// TIA Portal V20 export
// export: Created 2026-07-22T09:37:46.3128458Z, ExportSetting WithDefaults, DisplayName Totally Integrated Automation Portal, DisplayVersion V20, DisplayName TIA Portal Openness, DisplayVersion V20, DisplayName TIA Portal Version Control Interface, DisplayVersion V20, DisplayName STEP 7 Professional, DisplayVersion V20, DisplayName STEP 7 Safety, DisplayVersion V20, DisplayName WinCC Basic/Comfort/Advanced, DisplayVersion V20, DisplayName WinCC Professional, DisplayVersion V20, DisplayName WinCC Unified, DisplayVersion V20
TYPE "Valve_IO"
// stored: IsFailsafeCompliant false
   STRUCT
      Configured : Bool;
      OpenCmd : Bool;
      CloseCmd : Bool;
      LocalMode : Bool;
      Healthy : Bool;
      OpenFB : Bool;
      ClosedFB : Bool;
      OpenValve : Bool;
      CloseValve : Bool;
      TimerOpen : TON_TIME;
      TimerClose : TON_TIME;
   END_STRUCT;
END_TYPE
